GLOBALCONSTANTS NVS_Keys (* Global constants *)
  (* Standard: 61499-1 *)
  (* Version 1.0, 2025-02-12, franz *)
  VAR_GLOBAL CONSTANT
    KEY_GESAMTZAEHLER : STRING := 'Gesamtzaehler';
    KEY_GESAMTZIEL : STRING := 'Gesamtziel';
    KEY_TAGESZAEHLER : STRING := 'Tageszaehler';
    KEY_TAGESZIEL : STRING := 'Tagesziel';
  END_VAR
END_GLOBALCONSTANTS
